{attribute 'qualified_only'}
VAR_GLOBAL
	
	// HVAC_SEQ_28
	
	B28_STEP_1: BOOL;
	B28_STEP_2 : BOOL;
	B28_STEP_3 : BOOL;
	B28_STEP_4 : BOOL;
	B28_STEP_5 : BOOL;
	B28_STEP_6: BOOL;

END_VAR

(* stored: Version 1.1.0.1, ProductVersion 3.1.4024.13
   GVL SEQ: Id {8ed1fb12-3b79-4f3a-bc13-4cde9299cd12} *)
